{attribute 'GeneratedUsingTerminal: EK1122-0000-0018'}
{attribute addProperty BoxType "EK1122-0000-0018"}
{attribute addProperty Id "Beckhoff_APS4xxxsub_EK1100EK1100_1FC0878B2A_0001_APS4322_7000_0017APS4322_F59021E4274"}
{attribute addProperty CRC "2631628341"}
{attribute addProperty Size "276"}
TYPE Beckhoff_APS4xxxEK1122_9CDB7635 EXTENDS EK1122_1FC0878B :
STRUCT
	{attribute addProperty Name "Beckhoff_APS4xxxsub_EK1100"}
	{attribute addProperty PreviousPort "Beckhoff APS4xxxEK1122 : D"}
	Beckhoff_APS4xxxsub_EK1100 : EK1100_1FC0878B;
	{attribute addProperty Name "A_0001_APS4322_7000_0017"}
	{attribute addProperty PreviousPort "Beckhoff APS4xxxsub EK1100 : C"}
	A_0001_APS4322_7000_0017 : APS4322_F59021E4;
END_STRUCT
END_TYPE

(* stored: Version 1.2.0.0, ProductVersion 3.1.4024.9
   DUT Beckhoff_APS4xxxEK1122_9CDB7635: Id {927d6270-f961-4042-a557-6e92535207ae} *)
